// TIA Portal V20 export
TYPE "LER_typeVisionAlignResultData"
// stored: Access Published
   STRUCT
      tabFoldingMissingJudgementResult : Real;   // Tab Folding & Missing_Judgement Result (0:NONE,1:OK,2:NG)
      electrodeLengthJudgementResult : Real;   // Electrode length_Judgement Result (0:NONE,1:OK,2:NG)
      electrodeHeightJudgementResult : Real;   // Electrode length_Judgement Result (0:NONE,1:OK,2:NG)
      movementAmountAxisX1 : Real;   // X1축 이동량
      movementAmountAxisY1 : Real;   // Y1축 이동량
      movementAmountAxisY2 : Real;   // Y2축 이동량
      tabFoldingMissingReply : Real;   // Tab Folding & Missing_Reply [](1/1000)
      tabFoldingMissingUpperRangeReply : Real;   // Tab Folding & Missing_Upper Range Reply [](1/1000)
      tabFoldingMissingLowerRangeReply : Real;   // Tab Folding & Missing_Lower Range Reply [](1/1000)
      electrodeLengthReply : Real;   // Electrode length Reply [mm](1/1000)
      electrodeLengthUpperRangeReply : Real;   // Electrode length(1/1000) Upper Range Reply [mm](1/1000)
      electrodeLengthLowerRangeReply : Real;   // Electrode length(1/1000) Lower Range Reply [mm](1/1000)
      electrodeHeightReply : Real;   // Electrode height_Reply [mm](1/1000)
      electrodeHeightUpperRangeReply : Real;   // Electrode height(1/1000) Upper Range Reply [mm](1/1000)
      electrodeHeightLowerRangeReply : Real;   // Electrode height(1/1000) Lower Range Reply [mm](1/1000)
   END_STRUCT;
END_TYPE
